# B&R Automation Studio project Morozov_labs_semestr_7
Automation Studio 4.5.2.102

## Configuration Config1

### Hardware
```
4PP065_0571_P74 : 4PP065.0571-P74 v1.1.2.0
  Connector IF5:
    ActivateDevice = 1
    Mode = Manual
    InternetAddress = 10.0.1.10
    SubnetMask = 255.255.255.0
  ConfigurationID = labBR
  SimulationIPAddress = 10.0.1.10
```

## Logical view

### Library Logical/Libraries/MotorCtrl

#### MotorCtrl.fun
```iecst
{REDUND_ERROR} FUNCTION_BLOCK FB_Motor (* *) (*$GROUP=User,$CAT=User,$GROUPICON=User.png,$CATICON=User.png*)
	VAR_INPUT
		u : REAL; (*Входное напряжение, В*)
	END_VAR
	VAR_OUTPUT
		phi : REAL; (*Положение, рад*)
		w : REAL; (*Частота напряжения, об/мин*)
	END_VAR
	VAR
		dt : REAL := 0.003; (*Шаг расчёта, с*)
		ke : REAL; (*Постоянная ЭДС двигателя, В*мин/об*)
		Tm : REAL := 0.03; (*Электромеханическая постоянная времени, с*)
		integrator : FB_Integrator; (*Интегратор*)
	END_VAR
END_FUNCTION_BLOCK

{REDUND_ERROR} FUNCTION_BLOCK FB_Regulator (* *) (*$GROUP=User,$CAT=User,$GROUPICON=User.png,$CATICON=User.png*)
	VAR_INPUT
		e : REAL; (*Рассогласование между задающим воздействием и реальной скоростью вращения вала ДПТ, об/мин*)
	END_VAR
	VAR_OUTPUT
		u : REAL; (*Напряжение, подаваемое на вход ДПТ, В*)
	END_VAR
	VAR
		a : REAL;
		b : REAL;
		last_sum : REAL;
		sum : REAL;
		k_p : REAL := 0.0064; (*Пропорциональный коэффициент регулятора*)
		k_i : REAL := 0.16; (*Интегральный коэффициент регулятора*)
		integrator : FB_Integrator; (*Интегратор*)
		iyOld : REAL; (*Хранение предыдущего значения схемы противонакопления*)
		limited_sum : REAL;
		max_abs_value : REAL := 24; (*Граница блока ограничения, В*)
		dt : REAL := 0.003; (*Шаг расчёта, с*)
	END_VAR
END_FUNCTION_BLOCK

{REDUND_ERROR} FUNCTION_BLOCK FB_Integrator (* *) (*$GROUP=User,$CAT=User,$GROUPICON=User.png,$CATICON=User.png*)
	VAR_INPUT
		in : REAL; (*Выход интегрирующего звена*)
	END_VAR
	VAR_OUTPUT
		out : REAL; (*Вход интегрирующего звена*)
	END_VAR
	VAR
		dt : REAL := 0.003; (*Шаг расчёта, с*)
		prev_value : REAL; (*Предыдущее состояние*)
	END_VAR
END_FUNCTION_BLOCK
```

#### FB_Integrator.c
```c
#include <bur/plctypes.h>
#ifdef __cplusplus
	extern "C"
	{
#endif
	#include "MotorCtrl.h"
#ifdef __cplusplus
	};
#endif
/* TODO: Add your comment here */
void FB_Integrator(struct FB_Integrator* inst)
{
	inst->dt = d_t;
	inst->out = inst->dt * inst->in + inst->prev_value;
	inst->prev_value = inst->out;
}
```

#### FB_Motor.c
```c
#include <bur/plctypes.h>
#ifdef __cplusplus
	extern "C"
	{
#endif
	#include "MotorCtrl.h"
#ifdef __cplusplus
	};
#endif
/* TODO: Add your comment here */
void FB_Motor(struct FB_Motor* inst)
{
	REAL a = inst->u / inst->ke - inst->w;
	REAL b = a / inst->Tm;

	inst->integrator.in = b;
	FB_Integrator(&inst->integrator);

	inst->w = inst->integrator.out;
}
```

#### FB_Regulator.c
```c
#include <bur/plctypes.h>
#ifdef __cplusplus
	extern "C"
	{
#endif
	#include "MotorCtrl.h"
#ifdef __cplusplus
	};
#endif
/* TODO: Add your comment here */

void FB_Regulator(struct FB_Regulator* inst)
{
	inst->dt = d_t;
	inst->a = inst->e * inst->k_p;
	inst->b = inst->e * inst->k_i;

	inst->a = inst->a > inst->max_abs_value ? inst->max_abs_value : inst->a;
	inst->a = inst->a < -inst->max_abs_value ? -inst->max_abs_value : inst->a;

	inst->integrator.in = inst->b + inst->last_sum;
	FB_Integrator(&inst->integrator);

	inst->sum = inst->a + inst->integrator.out;
	inst->u = inst->sum;
	inst->u = inst->u > inst->max_abs_value ? inst->max_abs_value : inst->u;
	inst->u = inst->u < -inst->max_abs_value ? -inst->max_abs_value : inst->u;

	inst->last_sum = inst->u - inst->sum;
}
```

### Program Logical/Program

#### Variables.var
```iecst
VAR
	fb_motor4 : FB_Motor;
	fb_motor3 : FB_Motor;
	fb_motor2 : FB_Motor;
	fb_motor1 : FB_Motor;
	regulator : FB_Regulator;
	counter : USINT;
	speed : REAL;
	e : REAL;
	enable : BOOL;
END_VAR
```

#### Cyclic.c
```c
#include <bur/plctypes.h>

#ifdef _DEFAULT_INCLUDES
	#include <AsDefault.h>
#endif

void _CYCLIC ProgramCyclic(void)
{
	if(enable){
		if(counter == 250){
			speed = 0;
			counter = 0;
		}
		if(counter == 100){
			speed = 50;
		}
		counter++;

		regulator.e = speed - fb_motor1.w;
		FB_Regulator(&regulator);

		fb_motor1.u = regulator.u;
		FB_Motor(&fb_motor1);

		fb_motor2.u = speed*fb_motor2.ke;
		FB_Motor(&fb_motor2);

	}
}
```

#### Init.c
```c
#include <bur/plctypes.h>

#ifdef _DEFAULT_INCLUDES
	#include <AsDefault.h>
#endif

void _INIT ProgramInit(void)
{
	fb_motor1.Tm = 0.0149;
	fb_motor1.ke =  5.26;
	fb_motor1.u = 0.1;

	fb_motor2.Tm =  0.0149;
	fb_motor2.ke = 5.26;
	fb_motor2.u = 0.1;

	regulator.k_i = 0.86;
	regulator.k_p = 0.26;
	regulator.max_abs_value = 24.0;

	speed = 0;
	counter = 0;
}
```
